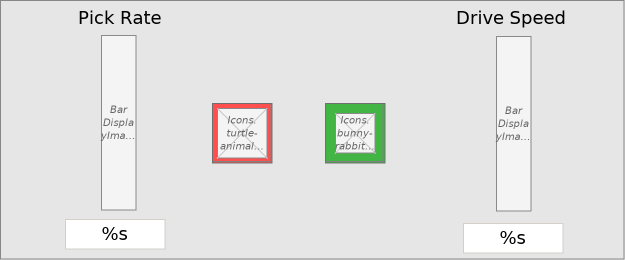
VISUALIZATION DriveControls  // 625x260
    Group (325,103 75x75)
        OnMouseClick: execute { HARV.DriveSys.AutoDriveSpeedCommand := HARV.DriveSys.AutoDriveSpeedCommand + 5; }
        Button (0,0 60x60)
        Image (10,10 40x40), image: Icons.bunny-rabbit-icon
    Group (212,103 75x75)
        OnMouseClick: execute { HARV.DriveSys.AutoDriveSpeedCommand := HARV.DriveSys.AutoDriveSpeedCommand - 5; }
        Button (0,0 60x60)
        Image (5,5 50x50), image: Icons.turtle-animal-icon
    Textfield (65,219 100x30), "%s"
    BarDisplayImage (101,35 35x175), style: BarDisplayImage-Gray, scale format: %.0f, scale 0..100
    BarDisplayImage (496,36 35x175), value: HARV.DriveSys.AutoDriveSpeedActual, style: BarDisplayImage-Gray, scale format: %.1f, scale 0..100
    Textfield (463,223 100x30), "%s", text variable: HARV.DriveSys.AutoDriveSpeedActual
    Textfield (436,3 150x30), "Drive Speed"
    Textfield (45,3 150x30), "Pick Rate"
END_VISUALIZATION

(* stored: Version 1.1.0.1, ProductVersion 3.1.4024.15
   Visu DriveControls: Id {edf9c3f4-94c9-4ee8-95d6-dc3c7c2f6e2a} *)
